(* PLC project PlainProject, Unknown Unnamed 1 *)
(* stored: creationDateTime 2023-09-14T08:06:45, modificationDateTime 2023-09-14T08:09:26 *)

PROGRAM program0
  VAR CONSTANT
    LocalVar0 : BOOL;
    LocalVar1 : BOOL;
  END_VAR

            LocalVar1 := LocalVar0;
          
END_PROGRAM

CONFIGURATION config
  RESOURCE resource1 ON PLC
    TASK task0(INTERVAL := T#20ms, PRIORITY := 0);
    PROGRAM instance0 WITH task0 : program0;
  END_RESOURCE
END_CONFIGURATION
